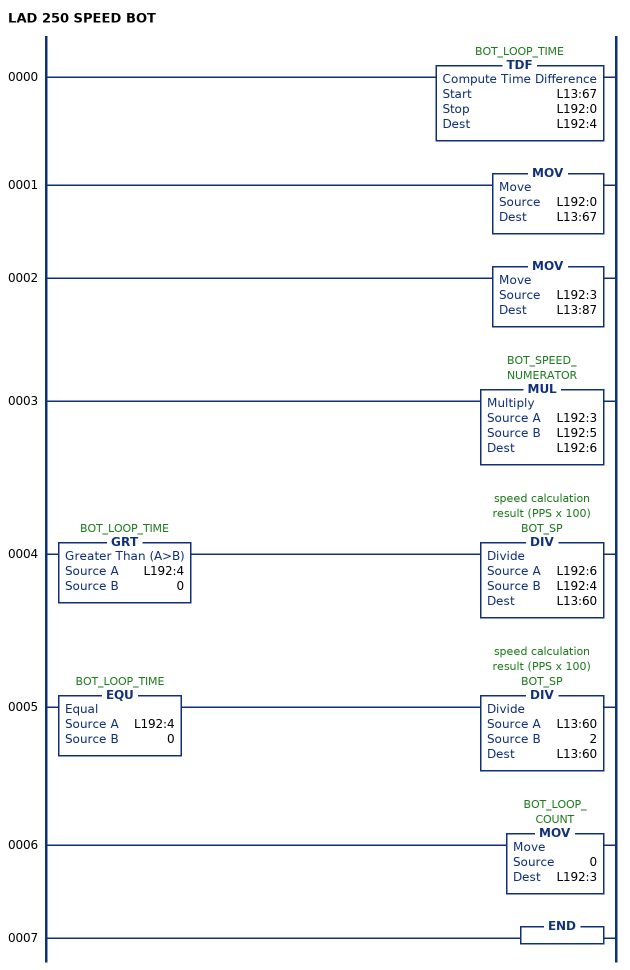
% Rung: 0 %
SOR TDF L13:67 L192:0 L192:4 EOR
%   L192:0  BOT_THIS_TIME  "rtc bot belt movement event time" %
%   L192:4  BOT_LOOP_TIME %
% Rung: 1 %
SOR MOV L192:0 L13:67 EOR
%   L192:0  BOT_THIS_TIME  "rtc bot belt movement event time" %
% Rung: 2 %
SOR MOV L192:3 L13:87 EOR
%   L192:3  BOT_LOOP_COUNT %
% Rung: 3 %
SOR MUL L192:3 L192:5 L192:6 EOR
%   L192:3  BOT_LOOP_COUNT %
%   L192:5  TKS_PER_SECOND %
%   L192:6  BOT_SPEED_NUMERATOR %
% Rung: 4 %
SOR GRT L192:4 0 DIV L192:6 L192:4 L13:60 EOR
%   L192:4  BOT_LOOP_TIME %
%   L192:6  BOT_SPEED_NUMERATOR %
%   L13:60  BOT_SP  "speed calculation result (PPS x 100)" %
% Rung: 5 %
SOR EQU L192:4 0 DIV L13:60 2 L13:60 EOR
%   L192:4  BOT_LOOP_TIME %
%   L13:60  BOT_SP  "speed calculation result (PPS x 100)" %
% Rung: 6 %
SOR MOV 0 L192:3 EOR
%   L192:3  BOT_LOOP_COUNT %
% Rung: 7 %
SOR END EOR

LADDER 251 "SPEED TOP"    % high speed %
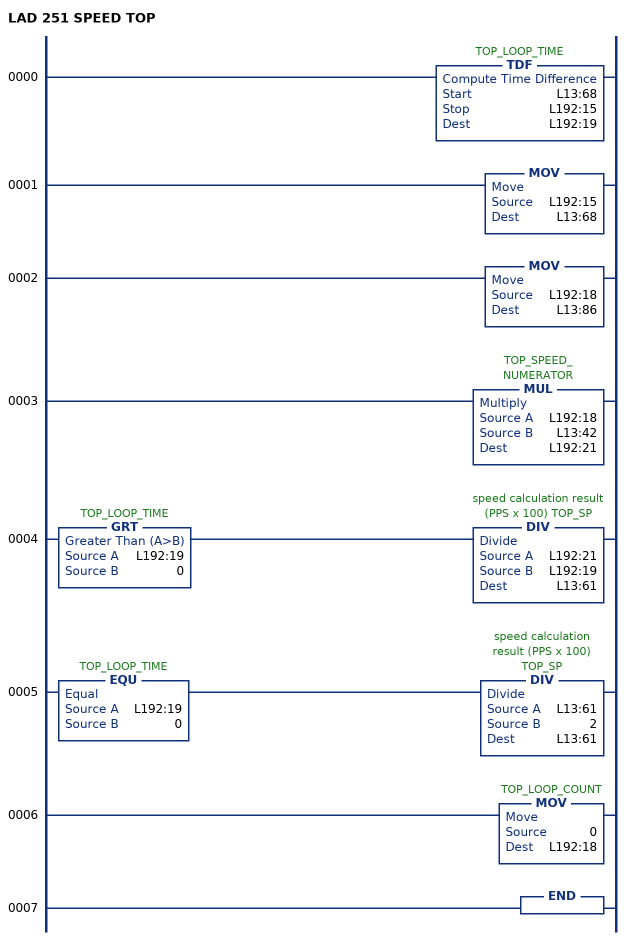
% Rung: 0 %
SOR TDF L13:68 L192:15 L192:19 EOR
%   L192:15  TOP_THIS_TIME  "rtc top belt movement event time" %
%   L192:19  TOP_LOOP_TIME %
% Rung: 1 %
SOR MOV L192:15 L13:68 EOR
%   L192:15  TOP_THIS_TIME  "rtc top belt movement event time" %
% Rung: 2 %
SOR MOV L192:18 L13:86 EOR
%   L192:18  TOP_LOOP_COUNT %
% Rung: 3 %
SOR MUL L192:18 L13:42 L192:21 EOR
%   L192:18  TOP_LOOP_COUNT %
%   L192:21  TOP_SPEED_NUMERATOR %
% Rung: 4 %
SOR GRT L192:19 0 DIV L192:21 L192:19 L13:61 EOR
%   L192:19  TOP_LOOP_TIME %
%   L192:21  TOP_SPEED_NUMERATOR %
%   L13:61  TOP_SP  "speed calculation result (PPS x 100)" %
% Rung: 5 %
SOR EQU L192:19 0 DIV L13:61 2 L13:61 EOR
%   L192:19  TOP_LOOP_TIME %
%   L13:61  TOP_SP  "speed calculation result (PPS x 100)" %
% Rung: 6 %
SOR MOV 0 L192:18 EOR
%   L192:18  TOP_LOOP_COUNT %
% Rung: 7 %
SOR END EOR

LADDER 252 "P BOT"    % high speed %
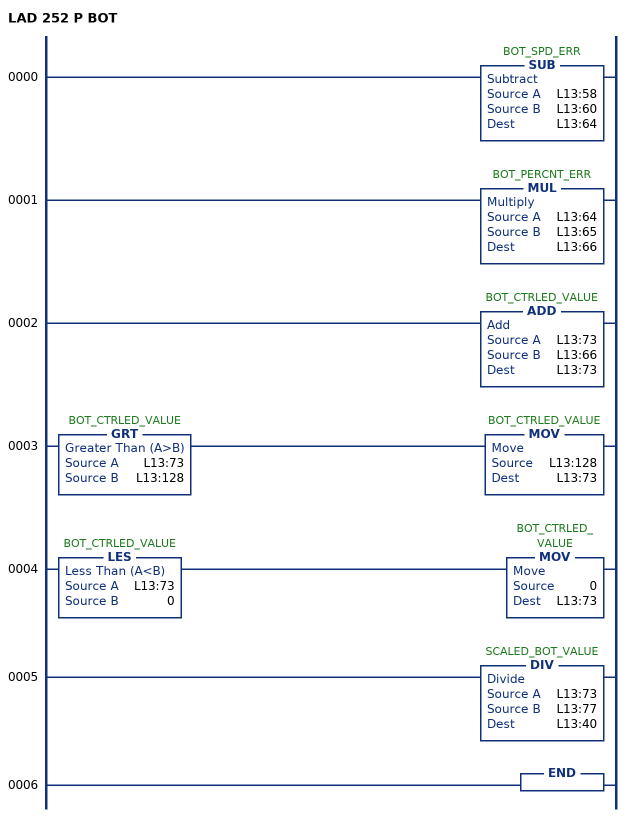
% Rung: 0 %
SOR SUB L13:58 L13:60 L13:64 EOR
%   L13:58  BOT_SPD_SETPOINT %
%   L13:60  BOT_SP  "speed calculation result (PPS x 100)" %
%   L13:64  BOT_SPD_ERR %
% Rung: 1 %
SOR MUL L13:64 L13:65 L13:66 EOR
%   L13:64  BOT_SPD_ERR %
%   L13:65  POS5SHIFT %
%   L13:66  BOT_PERCNT_ERR %
% Rung: 2 %
SOR ADD L13:73 L13:66 L13:73 EOR
%   L13:73  BOT_CTRLED_VALUE %
%   L13:66  BOT_PERCNT_ERR %
% Rung: 3 %
SOR GRT L13:73 L13:128 MOV L13:128 L13:73 EOR
%   L13:73  BOT_CTRLED_VALUE %
%   L13:128  "how much top has shifted since measurment" %
% Rung: 4 %
SOR LES L13:73 0 MOV 0 L13:73 EOR
%   L13:73  BOT_CTRLED_VALUE %
% Rung: 5 %
SOR DIV L13:73 L13:77 L13:40 EOR
%   L13:73  BOT_CTRLED_VALUE %
%   L13:40  SCALED_BOT_VALUE %
% Rung: 6 %
SOR END EOR

LADDER 253 "P TOP"    % high speed %
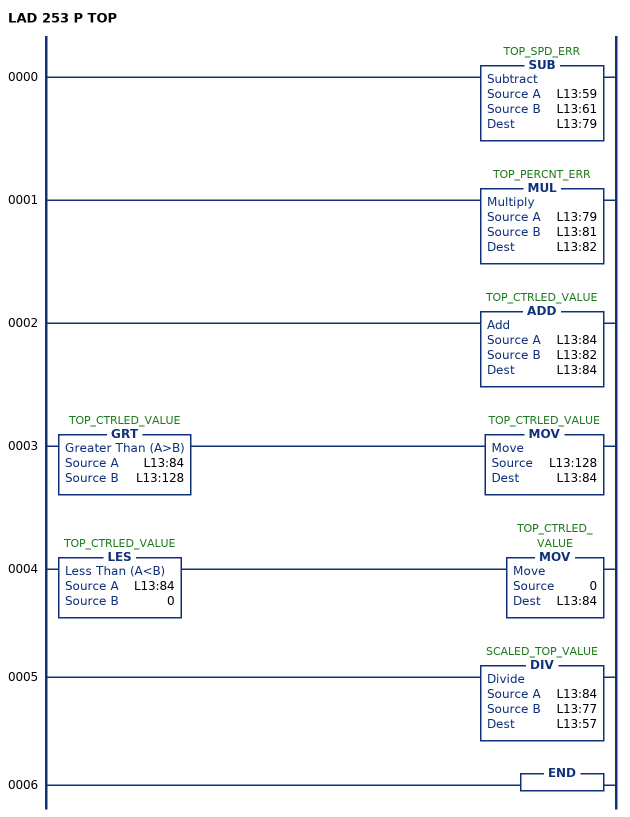
% Rung: 0 %
SOR SUB L13:59 L13:61 L13:79 EOR
%   L13:59  TOP_SPD_SETPOINT %
%   L13:61  TOP_SP  "speed calculation result (PPS x 100)" %
%   L13:79  TOP_SPD_ERR %
% Rung: 1 %
SOR MUL L13:79 L13:81 L13:82 EOR
%   L13:79  TOP_SPD_ERR %
%   L13:81  TOP_FDBK_RATIO %
%   L13:82  TOP_PERCNT_ERR %
% Rung: 2 %
SOR ADD L13:84 L13:82 L13:84 EOR
%   L13:84  TOP_CTRLED_VALUE %
%   L13:82  TOP_PERCNT_ERR %
% Rung: 3 %
SOR GRT L13:84 L13:128 MOV L13:128 L13:84 EOR
%   L13:84  TOP_CTRLED_VALUE %
%   L13:128  "how much top has shifted since measurment" %
% Rung: 4 %
SOR LES L13:84 0 MOV 0 L13:84 EOR
%   L13:84  TOP_CTRLED_VALUE %
% Rung: 5 %
SOR DIV L13:84 L13:77 L13:57 EOR
%   L13:84  TOP_CTRLED_VALUE %
%   L13:57  SCALED_TOP_VALUE %
% Rung: 6 %
SOR END EOR

LADDER 254 "TOTALCOUNT"
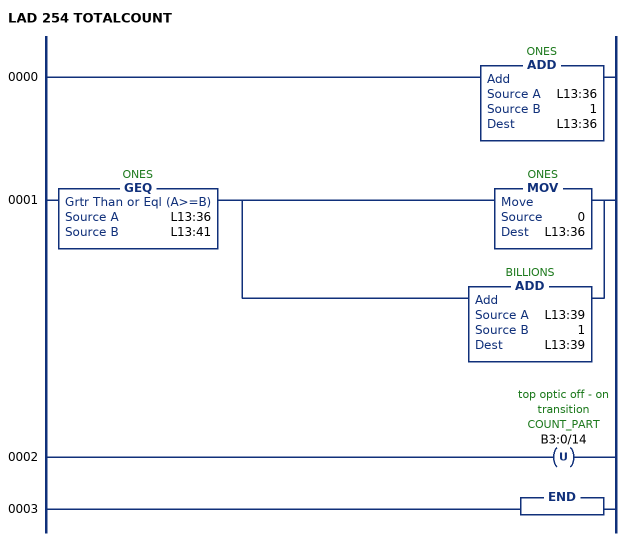
% Rung: 0 %
SOR ADD L13:36 1 L13:36 EOR
%   L13:36  ONES %
% Rung: 1 %
SOR GEQ L13:36 L13:41 BST MOV 0 L13:36 NXB ADD L13:39 1 L13:39 BND EOR
%   L13:36  ONES %
%   L13:41  "skipped count change in the last 3 seconds" %
%   L13:39  BILLIONS %
% Rung: 2 %
SOR OTU B3:0/14 EOR
%   B3:0/14  COUNT_PART  "top optic off - on transition" %
% Rung: 3 %
SOR END EOR

LADDER 255 "SAVED"
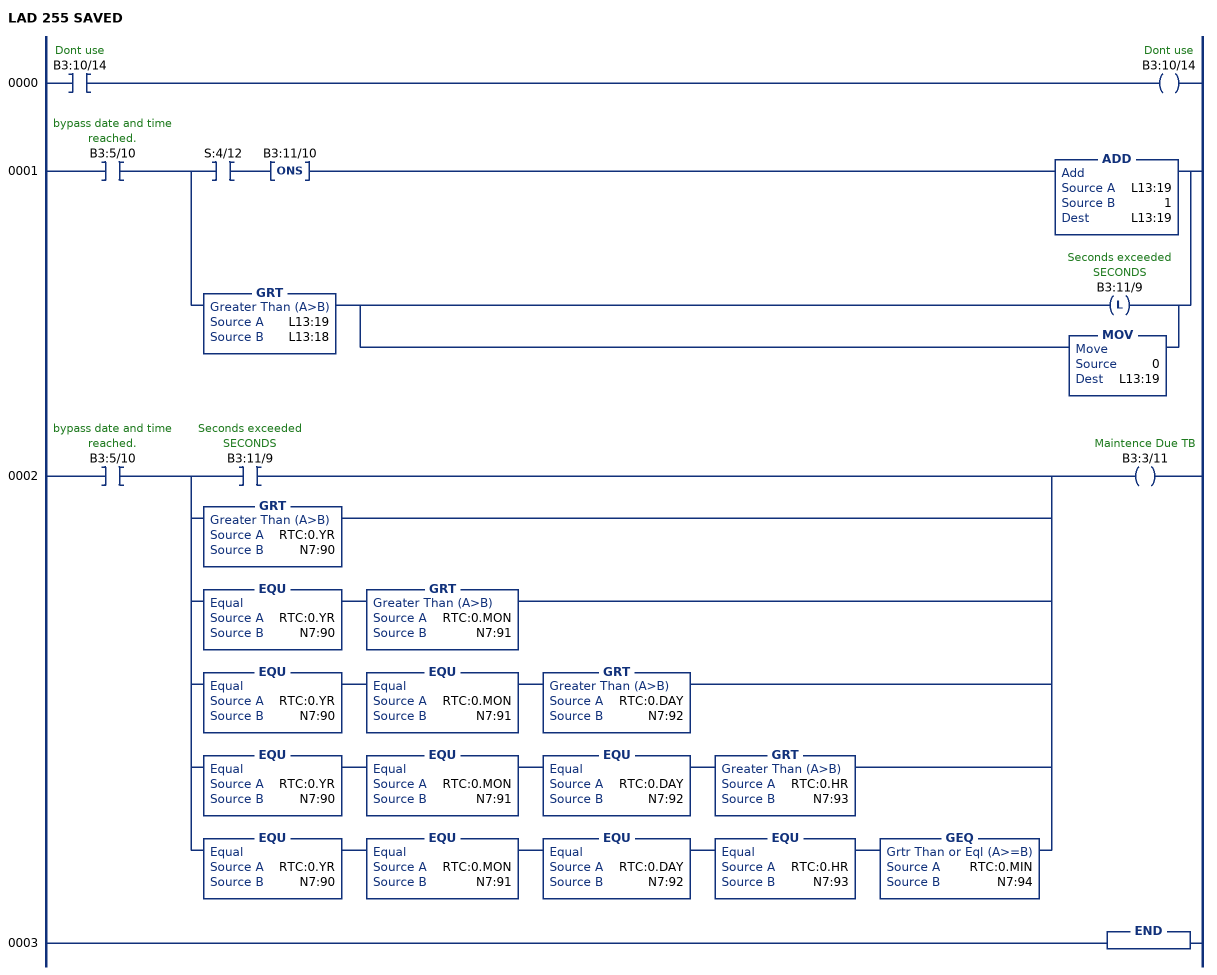
% Rung: 0 %
SOR XIC B3:10/14 OTE B3:10/14 EOR
%   B3:10/14  "Dont use" %
% Rung: 1 %
SOR XIC B3:5/10 BST XIC S:4/12 ONS B3:11/10 ADD L13:19 1 L13:19 NXB GRT L13:19 L13:18 BST OTL B3:11/9 NXB MOV 0 L13:19 BND BND EOR
%   B3:5/10  "bypass date and time reached." %
%   L13:18  MAX %
%   B3:11/9  SECONDS  "Seconds exceeded" %
% Rung: 2 %
SOR XIC B3:5/10 BST XIC B3:11/9 NXB GRT RTC:0.YR N7:90 NXB EQU RTC:0.YR N7:90 GRT RTC:0.MON N7:91 NXB EQU RTC:0.YR N7:90 EQU RTC:0.MON N7:91 GRT RTC:0.DAY N7:92 NXB EQU RTC:0.YR N7:90 EQU RTC:0.MON N7:91 EQU RTC:0.DAY N7:92 GRT RTC:0.HR N7:93 NXB EQU RTC:0.YR N7:90 EQU RTC:0.MON N7:91 EQU RTC:0.DAY N7:92 EQU RTC:0.HR N7:93 GEQ RTC:0.MIN N7:94 BND OTE B3:3/11 EOR
%   B3:5/10  "bypass date and time reached." %
%   B3:11/9  SECONDS  "Seconds exceeded" %
%   N7:90  RTC %
%   B3:3/11  TB  "Maintence Due" %
% Rung: 3 %
SOR END EOR

OTHER DOCUMENTED ADDRESSES
  B189:0/0  "change box"
  B189:0/9  "override boxing ok or not full signal"
  B189:0/11  "HMI force door close"
  B196:1/0  "Chute door is closed"
  B196:1/1  "control chute door"
  B196:1/13  "force box conveyor on"
  B196:3/0  "for hmi to continue production unlatched by hmi"
  HSC:0.0  "top"
  HSC:0.3/6  "Underflow interrupt"
  HSC:0.3/7  "Overflow interrupt"
  HSC:1.0  "bot"
  HSC:1.3/6  "Underflow interrupt"
  HSC:1.3/7  "Overflow interrupt"
  I:0.0/0  TOP_ENC
  I:0.0/2  CHUTE_OPTIC
  I:0.0/4  BOT_ENC
  I:0.0/10  "not used"
  I:0.1/4  "not used"
  I:0.1/5  "not used"
  I:0.1/6  "not used"
  I:0.1/7  "not used"
  I:0.1/8  "not used"
  I:0.1/9  "not used"
  I:0.1/10  "not used"
  I:0.1/11  "not used"
  I:0.1/12  "not used"
  I:0.1/13  "not used"
  I:0.1/14  "not used"
  I:0.1/15  "not used"
  I:0.2  "not used"
  I:0.2/3  "Packaging Conveyor full"
  I:0.2/4  "Packaging Conveyor Box in Position"
  I:0.3  "not used"
  I:0.4  "Spare Analog Input 1"
  I:0.5  "Spare Analog Input 2"
  I:0.6  "Spare Analog Input 3"
  I:2.0/0  FRONT_ESTOP
  I:2.0/1  REAR_ESTOP
  I:2.0/2  PACKAGER_CONNECTED
  I:2.0/3  BOX_CNV_NOT_FULL  "input turns off when box discharge full optics are blocked"
  I:2.0/4  BOX_NOT_IN_POS  "this input is on when a box is not in position"
  I:2.0/5  MCR
  I:2.0/6  MPCE  "primary safety relay on(e-stop)"
  I:2.0/7  MSCE  "secondary safety relay on(door) ce models only"
  I:2.0/8  FRONT_DOOR  "front door signal ce models only"
  I:2.0/9  REAR_DOOR  "rear door signal ce models only"
  I:2.0/10  MAINTENANCE_KEY_SW  "Maintenance Key Switch ce models only"
  I:2.0/11  "spare"
  I:2.0/12  "spare"
  I:2.0/13  FDER_PDL_SW  "Feeder Bowl Paddle Switch"
  I:2.0/14  "spare"
  I:2.0/15  TRACK_SENSOR  "Feeder Bowl Downtrack Sensor"
  L13:180  "maximum time between triggers"
  L13:181  "minimum okay time between triggers"
  L13:182  RATE_QUEUE_LIMIT
  L13:184  "intermediate i1 trig avg"
  L13:185  I1_TBT  "i1 average time between triggers"
  L13:186  "intermediate i5 trig avg"
  L13:187  I5_TBT  "i5 average time between triggers"
  L13:188  "intermediate i6 trig avg"
  L13:189  I6_TBT  "i6 average time between triggers"
  L13:190  "i1 timed q limit"
  L13:191  "i1 absolute q limit"
  L16:2  TRIG_DELAY_Q_MULTI
  L16:3  TRIG_DELAY_MIN_TIME
  L16:4  TRIG_DELAY_FLAT_RATE
  L16:5  CLEARTIME1  "time to clear tracking data"
  L16:6  CLEARTIME5
  L16:7  CLEARTIME6
  L16:8  PASS1PRTLOC
  L16:9  PASS1PROCESSTM
  L16:11  PASS5PROCESSTM
  L16:13  PASS6PROCESSTM
  L23:19  TOP_OPT_FAIL_CT
  L23:34  AIR_PRESSURE_FAULT
  L28:0  INS_1_TIME
  L29:0  INS_1_POS
  L30:0  INS_5_TIME
  L31:0  INS_5_POS
  L32:0  INS_6_TIME
  L33:0  INS_6_POS
  L192:1  BOT_LAST_TIME  "rtc bot belt previous movement event time"
  L192:2  BOT_CYCLE_TIME  "rtc bot belt time between events"
  L192:7  FROM_REAL  "distance from real part signal at optic location"
  L192:8  FROM_TRACKED  "distance from tracked part signal at optic location"
  L192:16  TOP_LAST_TIME  "rtc top belt previous movement event time"
  L192:17  TOP_CYCLE_TIME  "rtc top belt time between events"
  L199:5  ACQTM51
  L199:6  ACQTM52
  L199:7  ACQTM53
  L199:9  "ones"
  L199:10  "billions"
  L199:13  DUMP_LONG
  L199:15  ACQTM11
  L199:16  ACQTM12
  L199:17  ACQTM13
  L199:20  RESULTTM1
  L199:22  CLEARTIME5COUNT
  L199:23  CLEARTIME6COUNT
  L199:24  ACQTM61
  L199:25  ACQTM62
  L199:26  ACQTM63
  L199:27  TMSINCETRIG1
  L199:29  TMSINCETRIG5
  L199:30  TMSINCETRIG6
  L199:31  CLEARTIME1COUNT
  L199:32  RESULTTM5
  L199:33  RESULTTM6
  L199:34  MAXACQTM1
  L199:36  MAXACQTM6
  N15:5  INS_1_TRIG_LOC
  O:0.0/12  "not used"
  O:0.0/13  "not used"
  O:0.0/14  "not used"
  O:0.0/15  "not used"
  O:0.1  "not used"
  O:0.2  "not used"
  O:0.3  "not used"
  PFILE:6  "check for part jams"
  PFILE:10  "Bottom belt HSC"
  PFILE:12  "Top belt HSC"
  Q2:55  END_OF_MAIN
  Q5:94  END_OF_BELTS
  T20:0  "Trigger On Time"
  U:9  "slow data"
  U:24  "check skipped fail rate"
  U:28  "faults"
  U:29  "speed"
  U:30  "count"
  U:31  "rate calc"
  U:32  "boxer"
  U:33  "bulk pack"
  U:34  "customer boxing unit signals"
  U:35  "cleanup"

REVISION NOTES
  13: updated count reset
  14: added io moduals
  15: multiple steps toward new hmi integration
  21: test
  27: fix error if bulk pack and no boxing fallout were on

DATA TABLE (non-zero values as saved)
DATA B3
% B3:0 % 0X8000 0X1360 0X4000 0XA001 0X1EF5 0X0561 0X0038 0X0021 0X3F80 0X2558
% B3:10 % 0X20A0 0X2006 0X1005 0X0000 0X0000 0X0000 0X0000 0X0000 0X0000 0X0000
DATA T4
% .PRE .ACC %
% T4:1 % 150 0
% T4:2 % 400 0
% T4:3 % 222 0
% T4:4 % 1000 0
% T4:5 % 5 5
% T4:6 % 10 10
% T4:7 % 9000 0
% T4:8 % 20 15
% T4:9 % 50 11
% T4:10 % 200 200
% T4:11 % 333 0
% T4:12 % 100 102
% T4:13 % 250 0
% T4:14 % 666 0
% T4:15 % 1000 1001
% T4:16 % 400 0
% T4:17 % 100 42
% T4:18 % 5 0
% T4:19 % 300 0
% T4:20 % 200 0
% T4:21 % 200 0
% T4:22 % 200 0
% T4:23 % 250 0
% T4:24 % 666 0
% T4:25 % 666 0
% T4:26 % 666 0
% T4:27 % 250 0
% T4:28 % 250 0
% T4:29 % 5000 0
% T4:30 % 333 63
% T4:31 % 333 64
% T4:32 % 222 55
% T4:33 % 111 35
DATA C5
% .PRE .ACC %
% C5:0 % 32766 0
DATA R6
% .LEN .POS %
% R6:0 % 1250 0
% R6:1 % 1250 0
% R6:2 % 1024 0
% R6:3 % 1024 0
% R6:4 % 1250 0
% R6:5 % 1250 0
% R6:6 % 1713 0
% R6:7 % 1024 0
% R6:8 % 1024 0
% R6:9 % 3 0
% R6:10 % 1713 0
% R6:11 % 1713 0
% R6:12 % 10 0
% R6:13 % 10 0
% R6:14 % 10 0
% R6:15 % 10 0
% R6:16 % 1713 0
% R6:17 % 1713 0
% R6:18 % 1713 0
% R6:19 % 10 0
DATA N7
% N7:0 % 598 3 302 1000 18 400 0 500 500 500
% N7:10 % 1000 18 3000 2 20 20 1000 2000 50 1050
% N7:20 % 32767 111 10 333 333 46 48 0 48 250
% N7:30 % 666 5371 150 0 0 376 24 49 1 48
% N7:40 % 0 40 0 40 32767 482 388 632 1257 8
% N7:50 % 7 16 8 16 17 245 19659 19659 32766 18
% N7:60 % 1713 1713 1713 1021 1034 1024 4999 5 400 400
% N7:70 % 100 200 300 400 90 190 290 390 4735 1099
% N7:80 % 0 0 397 780 832 844 44 27 0 3
% N7:90 % 2011 4 4 12 1 44 24 222 111 12
% N7:100 % 1003 90 110 100 175 25 0 0 0 245
DATA F8
% F8:0 % 6 1 23807 499 0.23807
% F8:5 % 0 0 500 1.9 2
% F8:10 % 1 0.08897486 3058 101 63.26563
% F8:15 % 37.73437 4040 2 0 0
% F8:20 % 0 0.02 0 1 0
% F8:25 % 0 932781 0.222 279.6551 848597
% F8:30 % 0 170 0.03 38 852060
% F8:35 % 0 0 0 0 77
% F8:40 % 101 37.73437 0 100 1
% F8:45 % 1 2 0.21455 0 0
% F8:50 % 0 0 1 0 1
% F8:55 % 2000000 -221 0 0 0
% F8:95 % 0 0 0 492 4.92
DATA B12
% B12:0 % 0X3540 0X0000 0X0000 0X0000 0X0000 0X0000 0X0000 0X0000 0X0000 0X0000
DATA L13
% L13:0 % 14895 15868 0 1658944 1883814
% L13:5 % 78 15570 0 26000 1634961
% L13:10 % 1578031 549963602 0 15 90
% L13:15 % 2136772161 -2147483648 2147483647 2147483647 82058
% L13:20 % 1326931947 1879169009 777 367734 100
% L13:25 % 153441500 49 684 0 2135432029
% L13:30 % 1339362 1386 1020000 409312962 444
% L13:35 % 27 1889597 1 78 0
% L13:40 % 1340 1000000000 1000000 1195891046 2135928652
% L13:45 % 1195890969 9025 0 58 1612026828
% L13:50 % 843550 27363 2079664181 0 0
% L13:55 % 30666 136347 1402 3000 3000
% L13:60 % 3001 3003 58 600 -1
% L13:65 % 3 -3 480003663 480003660 -942969229
% L13:70 % 1875789486 31 764408719 133958 1612026828
% L13:75 % 74593915 60 100 2079664212 -3
% L13:80 % 31 3 -9 0 140177
% L13:85 % 255209 152 152 0 5
% L13:90 % 10 5 1889597 10 2135928681
% L13:95 % 12 338 0 409313968 1402
% L13:100 % 2147483647 6353502 900 3 338
% L13:105 % 1402 9 1326019172 133426 1326019166
% L13:110 % 6 30 25 1328950220 1878913819
% L13:115 % 1878913822 3 2 1878913820 2
% L13:120 % 13 82 25 30 47
% L13:125 % 0 1875789486 2147483647 3276500 550218823
% L13:130 % 2 2 0 999999 0
% L13:135 % 0 0 255221 5 1
% L13:140 % 0 5 36 21 50
% L13:145 % 5 5 5 5 12
% L13:150 % 1 7 133420 -133420 549963602
% L13:155 % 0 -9 0 0 4589052
% L13:160 % 24 29 24 29 24
% L13:165 % 1878913905 1612027195 1878913905 1612027195 7
% L13:170 % 6184 270 117 1200 4700
% L13:175 % 4 40 42 23 38
% L13:180 % 176247033 25 99000 52866 644409
% L13:185 % 64 916459 92 627156 63
% L13:190 % 4 5 0 0 0
DATA F14
% F14:0 % 1.32889e-38 5747.126 1550 1550 1638.3
% F14:5 % 1638.3 1638.3 1638.3 0 0
DATA N15
% N15:0 % 385 500 685 375 320 128 100 1184 300 10
% N15:10 % 71 887 0 0 0 0 1356 0 0 0
DATA L16
% L16:0 % 10 100 11 0 20
% L16:5 % 250 5000 5000 182 19
% L16:10 % 1256 18 2045 6599584 98
% L16:15 % 99 0 0 0 0
DATA L19
% L19:0 % 2135926699 2135926823 2135927163 2135927385 2135927654
% L19:5 % 2135927871 2135928109 2135928380 2135432029 2135432276
% L19:10 % 2135432517 2135439204 2135439468 2135439686 2135439899
% L19:15 % 2135440159 2135440286 0 0 0
DATA L20
% L20:0 % 2135158985 2135159229 2135159527 2135215738 2135215966
% L20:5 % 2135216198 2135216436 2135216658 2135216896 2135217154
% L20:10 % 2135217402 2135256885 2135257123 2135257347 2135257580
% L20:15 % 2135257835 2135297623 2135297882 2135298135 2135298363
% L20:20 % 2135298577 2135298859 2135324259 2135324476 2135324768
% L20:25 % 2135431555 2135431787 2135431990 2135432305 2135432549
% L20:30 % 2135432791 2135439478 2135439745 2135439961 2135440175
% L20:35 % 2135440432 2135440561 2135926973 2135927097 2135927437
% L20:40 % 2135927660 2135927926 2135928144 2135928382 2135928652
% L20:45 % 2135157932 2135158145 2135158274 2135158532 2135158790
DATA L21
% L21:0 % 1878681144 1878681218 1878681308 1878698308 1878698377
% L21:5 % 1878698447 1878698519 1878698586 1878698658 1878698736
% L21:10 % 1878698811 1878710749 1878710821 1878710889 1878710959
% L21:15 % 1878711036 1878723068 1878723146 1878723223 1878723292
% L21:20 % 1878723357 1878723442 1878731124 1878731190 1878731278
% L21:25 % 1878763573 1878763643 1878763705 1878763800 1878763874
% L21:30 % 1878763947 1878765969 1878766050 1878766115 1878766180
% L21:35 % 1878766258 1878766297 1878913397 1878913434 1878913537
% L21:40 % 1878913604 1878913685 1878913751 1878913823 1878913905
% L21:45 % 1878680825 1878680890 1878680929 1878681007 1878681085
DATA L22
% L22:0 % 1180145959 1180146075 1180147227 1180147343 1180147458
% L22:5 % 1180147574 1181268908 1181269023 1181269138 1181269254
% L22:10 % 1181270406 1181270521 1181270637 1181270752 1181324205
% L22:15 % 1181363998 1181733647 1181735250 1181735608 1195874847
% L22:20 % 1195889455 1195889571 1195889687 1195889805 1195890969
% L22:25 % 1195891087 1195891202 1195891319 1179403719 1179403834
% L22:30 % 1179403948 1179404063 1180001030 1180001144 1180001261
% L22:35 % 1180001375 1180002530 1180002645 1180002761 1180002876
% L22:40 % 1180076101 1180076215 1180076332 1180076448 1180077599
% L22:45 % 1180077714 1180077830 1180077947 1180145729 1180145845
DATA L23
% L23:0 % 1687263579 1687263591 1687263707 1687263719 1687263730
% L23:5 % 1687263742 1687376771 1687376783 1687376794 1687376806
% L23:10 % 1687376922 1687376934 1687376945 1687376957 1687382345
% L23:15 % 1687386356 1687423616 1687423778 1687423814 1689725663
% L23:20 % 1689728606 1689728630 1689728653 1689728677 1689728913
% L23:25 % 1689728937 1689728961 1689728985 1687193515 1687193526
% L23:30 % 1687193538 1687193549 1687248971 1687248983 1687248994
% L23:35 % 1687249006 1687249123 1687249134 1687249146 1687249158
% L23:40 % 1687256538 1687256550 1687256561 1687256573 1687256689
% L23:45 % 1687256700 1687256712 1687256724 1687263556 1687263568
DATA L30
% L30:0 % 1182049462 1182049808 1182051193 1182051539 1182052915
% L30:5 % 1182053261 1182054645 1182054993 1182056375 1182056721
% L30:10 % 1182058100 1182058446 1182059829 1182060175 1182061560
% L30:15 % 1182061903 1182063290 1182063634 1182065017 1182065359
% L30:20 % 1182066737 1182067083 1182068465 1182068807 1182070191
% L30:25 % 1182070535 1182071922 1182072267 1182073653 1182073996
% L30:30 % 1182075380 1182075720 1182077097 1182077441 1182078825
% L30:35 % 1182079168 1182080545 1182080893 1182082278 1182082619
% L30:40 % 1182084005 1182084349 1182085737 1182086077 1182087456
% L30:45 % 1182087802 1195889348 1195889691 1195891046 1195891384
DATA L31
% L31:0 % 1687473526 1687473596 1687473874 1687473944 1687474221
% L31:5 % 1687474291 1687474573 1687474644 1687474922 1687474992
% L31:10 % 1687475271 1687475341 1687475617 1687475687 1687475965
% L31:15 % 1687476035 1687476312 1687476382 1687476662 1687476731
% L31:20 % 1687477006 1687477076 1687477354 1687477423 1687477700
% L31:25 % 1687477770 1687478051 1687478121 1687478397 1687478467
% L31:30 % 1687478747 1687478816 1687479092 1687479162 1687479443
% L31:35 % 1687479513 1687479791 1687479862 1687480143 1687480212
% L31:40 % 1687480489 1687480559 1687480839 1687480908 1687481184
% L31:45 % 1687481254 1689728584 1689728654 1689728929 1689728998
DATA L32
% L32:0 % 2075102604 2075102974 2075107193 2075107642 2075107974
% L32:5 % 2075108185 2075287746 2076696670 2076697006 2076698352
% L32:10 % 2076698688 2076773100 2076773436 2076773772 2076774108
% L32:15 % 2076774445 2076774781 2076775117 2076850718 2076851054
% L32:20 % 2076852398 2076852734 2076891699 2076892158 2076892836
% L32:25 % 2077491707 2077519818 2077582506 2077601288 2077643908
% L32:30 % 2077655050 2077671855 2077684309 2079660687 2079662159
% L32:35 % 2079662496 2079662833 2079663170 2079663506 2079663843
% L32:40 % 2079664181 2075100650 2075100865 2075101132 2075101291
% L32:45 % 2075101510 2075101814 2075102138 2075102302 2075102488
DATA L33
% L33:0 % 1874853135 1874853247 1874854523 1874854659 1874854759
% L33:5 % 1874854823 1874909124 1875297777 1875297777 1875297777
% L33:10 % 1875297777 1875297777 1875297777 1875297777 1875297777
% L33:15 % 1875297777 1875297777 1875297777 1875297777 1875297777
% L33:20 % 1875297777 1875297777 1875297884 1875297997 1875298187
% L33:25 % 1875419590 1875425257 1875437897 1875441686 1875450277
% L33:30 % 1875452523 1875455910 1875458421 1875788430 1875788875
% L33:35 % 1875788977 1875789079 1875789181 1875789283 1875789384
% L33:40 % 1875789486 1874852544 1874852609 1874852690 1874852738
% L33:45 % 1874852804 1874852896 1874852994 1874853044 1874853100
DATA B38
% B38:10 % 0X0000 0X0000 0X0000 0X0000 0X0000 0X0000 0X0000 0X0000 0XE000 0XFFFE
% B38:20 % 0X007C 0X2000 0X0000 0X0000 0X0000 0X0000 0X0000 0X0000 0X0000 0X0000
% B38:60 % 0X0000 0X0000 0X0080 0X8800 0X0003 0X0000 0X0FFF 0X0000 0X0000 0X0000
% B38:120 % 0X0000 0X0000 0X0000 0X0000 0X0000 0X0000 0X0000 0X0002
DATA B40
% B40:10 % 0X0000 0X0000 0X0000 0X0000 0X0000 0X0000 0X0000 0X0000 0XE000 0XFFFE
% B40:20 % 0X007C 0X2000 0X0000 0X0000 0X0000 0X0000 0X0000 0X0000 0X0000 0X0000
% B40:60 % 0X0000 0X0000 0X0080 0X8800 0X0003 0X0000 0X0FFF 0X0000 0X0000 0X0000
% B40:120 % 0X0000 0X0000 0X0000 0X0000 0X0000 0X0000 0X0000 0X0002
DATA L192
% L192:0 % 480169933 266932201 5055 41 50890
% L192:5 % 1000000 153000000 999 999 8
% L192:10 % 0 192814634 0 78 17
% L192:15 % 480170100 332250347 860888 42 50708
% L192:20 % 180 152000000 0 0 0
DATA B196
% B196:0 % 0X0836 0X9FF6 0X0005 0X0000 0X0000 0X0000 0X0000 0X0000 0X0000 0X0000
% B196:30 % 0XE800 0X9BFF 0XEBFF 0XFFDF 0XFFFF 0X0000 0X0000 0X0000 0X0000 0X0000
DATA L199
% L199:0 % 1 0 0 0 0
